// TwinCAT 3 PLC project MQTT_2
// ProgramVersion: 3.1.4023.0
// libraries:
//   Tc2_Standard, * (Beckhoff Automation GmbH)
//   Tc2_System, * (Beckhoff Automation GmbH)
//   Tc2_Utilities, * (Beckhoff Automation GmbH)
//   Tc3_IotBase, * (Beckhoff Automation GmbH)
//   Tc3_Module, * (Beckhoff Automation GmbH)
// project tree:
//   / PlcTask.TcTTO
//   POUs/ MAIN.TcPOU, testClient1.TcPOU, testClient2.TcPOU
// (motion and I/O tree: see PLC project ftp)
// real-time tasks:
//   TASK PlcTask: cycle T#10ms, priority 20, ADS port 350
//   TASK PlcTask1: cycle T#10ms, priority 21, ADS port 351
//   TASK PlcTask2: cycle T#10ms, priority 22, ADS port 352
//   TASK PlcTask3: cycle T#10ms, priority 23, ADS port 353
//   TASK PlcTask4: cycle T#10ms, priority 24, ADS port 354
//   TASK PlcTask5: cycle T#10ms, priority 25, ADS port 355
//   TASK PlcTask6: cycle T#10ms, priority 26, ADS port 356

CONFIGURATION MQTT_2
    RESOURCE PLC ON TwinCAT3
        TASK PlcTask(INTERVAL := T#10ms, PRIORITY := 26);
        PROGRAM MAIN WITH PlcTask : MAIN;
    END_RESOURCE
END_CONFIGURATION

// ---- POUs/MAIN.TcPOU
PROGRAM MAIN
VAR
END_VAR

//testClient1();
testClient2();

END_PROGRAM

// ---- POUs/testClient2.TcPOU
PROGRAM testClient2

VAR_INPUT
	bSetParameter : BOOL := TRUE;
END_VAR

VAR
	FB_IotMqttClient : FB_IotMqttClient;
	FB_IotMqttMessageQueue : FB_IotMqttMessageQueue;
	FB_IotMqttMessage : FB_IotMqttMessage;
	
	bSubscribed    : BOOL;
	sTopicSub      : STRING(255) := '$$SYS/broker/clients/connected';
    {attribute 'TcEncoding':='UTF-8'}
    sTopicRcv      : STRING(255);
    {attribute 'TcEncoding':='UTF-8'}
    sPayloadRcv    : STRING(5);
	fbTimer: TON;
	i: UINT;
	sPayloadPub: STRING(255);
END_VAR

IF bSetParameter THEN
	FB_IotMqttClient.sHostName:= 'broker.hivemq.com';
	FB_IotMqttClient.nHostPort:= 1883;
	FB_IotMqttClient.ipMessageQueue:= FB_IotMqttMessageQueue;
	bSetParameter:= FALSE;
END_IF

FB_IotMqttClient.Execute(TRUE);

IF FB_IotMqttClient.bConnected THEN
    fbTimer(IN:=TRUE);
    IF fbTimer.Q THEN // publish new payload every second
        fbTimer(IN:=FALSE);
        i := i + 1;
        sPayloadPub := 'Landen';
        FB_IotMqttClient.Publish( sTopic:= 'PXLcommunicationRX', 
                                  pPayload:= ADR(sPayloadPub), nPayloadSize:= LEN2(ADR(sPayloadPub))+1, 
                                  eQoS:= TcIotMqttQos.AtMostOnceDelivery, bRetain:= FALSE, bQueue:= FALSE );
    END_IF
END_IF

END_PROGRAM

// ---- POUs/testClient1.TcPOU
PROGRAM testClient1

VAR_INPUT
	bSetParameter : BOOL := TRUE;
END_VAR

VAR
	FB_IotMqttClient : FB_IotMqttClient;
	FB_IotMqttMessageQueue : FB_IotMqttMessageQueue;
	FB_IotMqttMessage : FB_IotMqttMessage;
	
	bSubscribed    : BOOL;
	sTopicSub      : STRING(255) := 'testTopic';
    {attribute 'TcEncoding':='UTF-8'}
    sTopicRcv      : STRING(255);
    {attribute 'TcEncoding':='UTF-8'}
    sPayloadRcv    : STRING(50);
END_VAR

IF bSetParameter THEN
	FB_IotMqttClient.sHostName:= 'broker.hivemq.com';
	FB_IotMqttClient.nHostPort:= 1883;
	FB_IotMqttClient.ipMessageQueue:= FB_IotMqttMessageQueue;
	bSetParameter:= FALSE;
END_IF

FB_IotMqttClient.Execute(TRUE);

IF FB_IotMqttClient.bConnected THEN
	IF NOT bSubscribed THEN
		bSubscribed := FB_IotMqttClient.Subscribe(sTopic:=sTopicSub, eQoS:=TcIotMqttQos.AtMostOnceDelivery);
	END_IF
END_IF

IF FB_IotMqttMessageQueue.nQueuedMessages > 0 THEN
	IF FB_IotMqttMessageQueue.Dequeue(fbMessage:=FB_IotMqttMessage) THEN
		FB_IotMqttMessage.GetTopic(pTopic:=ADR(sTopicRcv), nTopicSize:=SIZEOF(sTopicRcv) );
		FB_IotMqttMessage.GetPayload(pPayload:=ADR(sPayloadRcv), nPayloadSize:=SIZEOF(sPayloadRcv), bSetNullTermination:=FALSE);
	END_IF
END_IF

END_PROGRAM
